// TIA Portal V20 export
ORGANIZATION_BLOCK "MC_PreInterpolator"   // OB68, LAD, PreInterpolator
// stored: SetENOAutomatically false
   VAR_INPUT
      Initial_Call : Bool;
      PIP_Input : Bool;
      PIP_Output : Bool;
      IO_System : USInt;
      Event_Count : Int;
      Reduction : UInt;
      CycleTime : UDInt;
   END_VAR
BEGIN
END_ORGANIZATION_BLOCK
